Omron Sysmac Studio project nx1p2_hmi_weintek (Sysmac Studio 1.45.1.64010, StandardProject)

# Controller new_Controller_0: NX1P2-9024DT version 1.40
Task PrimaryTask (priority 4, period or condition 2000): Program0

VAR_GLOBAL
    NX1P2_IN_0 : BOOL;  (* at BuiltInIO://cpu/#0/Input_Bit_00; published *)
    NX1P2_IN_1 : BOOL;  (* at BuiltInIO://cpu/#0/Input_Bit_01; published *)
    NX1P2_OUT_0 : BOOL;  (* at BuiltInIO://cpu/#0/Output_Bit_00; published *)
END_VAR

PROGRAM Program0
VAR_EXTERNAL
    NX1P2_IN_0 : BOOL;
    NX1P2_IN_1 : BOOL;
    NX1P2_OUT_0 : BOOL;
END_VAR

(* Section Section0: ladder, written here as Structured Text *)

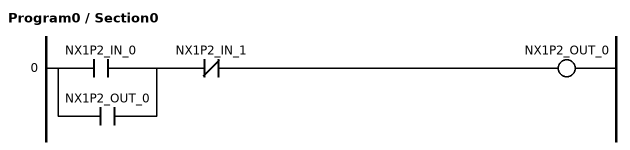
(* Rung 0 *)
NX1P2_OUT_0 := (NX1P2_IN_0 OR NX1P2_OUT_0) AND NOT NX1P2_IN_1;
END_PROGRAM